Staubli VAL3: logandpopMsg.pgx

program logandpopMsg(string x_sString (dimensions=1), bool& x_bBool (dimensions=1))
begin
  if x_bBool
    popUpMsg(x_sString)
    logMsg(x_sString)
    x_bBool=false
  endIf
  call massage(x_sString)
  delay(0.2)
end
